FUNCTION_BLOCK FB_LightGroup
VAR
	CurrentSizeOfLightGroup		: USINT := 0;
	aLights						: ARRAY[0..MAIN.MAXIMUM_NUMBER_OF_LIGHTS-1] OF I_LightBase;
	nCounter					: USINT;
	
	bIsOn						: bool := false;
END_VAR

// import all lights from main

FOR nCounter := 0 TO CurrentSizeOfLightGroup - 1 DO
	IF aLights[nCounter].State THEN
		bIsOn := TRUE;
		EXIT;
	ELSE
		IF nCounter = CurrentSizeOfLightGroup - 1 THEN
			bIsOn := FALSE;
		END_IF
	END_IF
END_FOR

METHOD ImportLight : BOOL
VAR_INPUT
	iLight		: I_LightBase;
END_VAR
aLights[CurrentSizeOfLightGroup]	:= iLight;
CurrentSizeOfLightGroup := CurrentSizeOfLightGroup + 1;
iLight.ID := CurrentSizeOfLightGroup;
END_METHOD

METHOD SetBrightness
VAR_INPUT
	nBrightness	: USINT;
END_VAR
VAR
	nCounter: USINT;
	iBrightness	: I_LightDimmable;
END_VAR
IF aLights[nCounter] <> 0 THEN
	FOR nCounter := 0 TO CurrentSizeOfLightGroup-1 DO
		IF __QUERYINTERFACE(aLights[nCounter], iBrightness) THEN
			iBrightness.Brightness := nBrightness;
		END_IF
	END_FOR
END_IF
END_METHOD

METHOD TurnOFF
VAR
	nCounter	: USINT;
END_VAR
FOR nCounter := 0 TO CurrentSizeOfLightGroup-1	DO
	aLights[nCounter].State := FALSE;
END_FOR
END_METHOD

METHOD TurnON
VAR
	nCounter	: USINT;
END_VAR
FOR nCounter := 0 TO CurrentSizeOfLightGroup-1	DO
	aLights[nCounter].State := TRUE;
END_FOR
END_METHOD

END_FUNCTION_BLOCK

(* stored: Version 1.1.0.1, ProductVersion 3.1.4024.12
   POU FB_LightGroup: Id {19f25f1a-18d9-4cfd-896f-2f3b9d975e5f}, SpecialFunc None
   Method ImportLight: Id {2725495e-2852-49f7-bfd1-5cb3d4b771d3}
   Method SetBrightness: Id {329af244-c0ff-48dc-8122-9466cb7fdce5}
   Method TurnOFF: Id {a83d100f-c41b-4130-8ead-8a196732aed6}
   Method TurnON: Id {a96c4366-e498-4aa9-b43c-4616a71ba20e} *)
